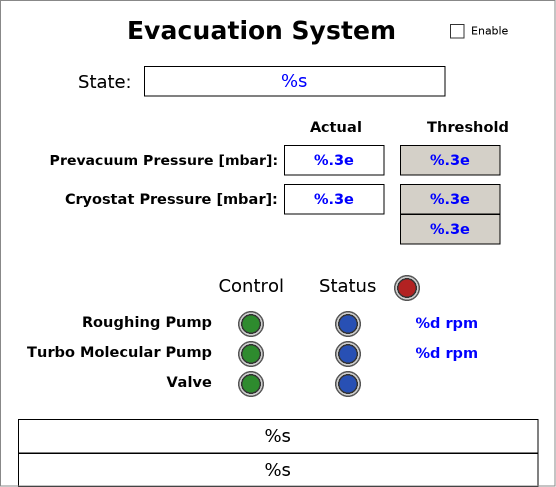
VISUALIZATION GUI_TEMPLATE_CRYO_EVAC_BASE  // 556x487
VAR_IN_OUT
	m_Instance:	FB_CRYO_EVAC_BASE;
	m_bEnable:	BOOL;
END_VAR
    Rectangle (144,66 301x30), "%s", text variable: m_Instance.stat.sState
    Lamp1 (236,309 30x30), variable: m_Instance.ctrl.bEnable_RP, style: Lamp-Lamp1-Green
    Rectangle (15,307 200x30), "Roughing Pump"
    Lamp1 (236,339 30x30), variable: m_Instance.ctrl.bEnable_TP, style: Lamp-Lamp1-Green
    Rectangle (15,337 200x30), "Turbo Molecular Pump"
    Lamp1 (236,369 30x30), variable: m_Instance.ctrl.bEnable_Valve, style: Lamp-Lamp1-Green
    Rectangle (15,367 200x30), "Valve"
    Rectangle (18,419 520x34), "%s", tooltip "Error description", text variable: m_Instance.stat.sErrorText
    Checkbox (448,16 108x30), "Enable", variable: m_bEnable
    Rectangle (56,67 84x30), "State:"
    Rectangle (299,271 98x30), "Status"
    Rectangle (284,145 100x30), "%.3e", tooltip "Prevacuum pressure [mbar]", text variable: m_Instance.prevac.stat.lrPressure
    Rectangle (400,145 100x30), "%.3e", tooltip "Prevacuum pressure threshold [mbar]", text variable: m_Instance.cfg.lrThld_Prevac
    Rectangle (284,184 100x30), "%.3e", tooltip "Cryo pressure [mbar]", text variable: m_Instance.in_lrCryoPressure
    Rectangle (400,184 100x30), "%.3e", tooltip "Pressure threshold for safe start of Turbo Pump [mbar]", text variable: m_Instance.cfg.lrThld_TP_SafeStartPressure
    Rectangle (400,214 100x30), "%.3e", tooltip "Pressure threshold for safe opening of the pre-vacuum valve [mbar]", text variable: m_Instance.cfg.lrThld_Valve_SafeOpenPressure
    Rectangle (51,145 230x30), "Prevacuum Pressure [mbar]:"
    Rectangle (51,184 230x30), "Cryostat Pressure [mbar]:"
    Rectangle (307,112 232x30), "Actual Threshold"
    Lamp1 (333,309 30x30), tooltip "If ON, Pump is Running", variable: m_Instance.stat.bRootPumpON, style: Lamp-Lamp1-Blue
    Lamp1 (333,339 30x30), tooltip "If ON, Pump is Running", variable: m_Instance.stat.bTurboPumpON, style: Lamp-Lamp1-Blue
    Lamp1 (333,369 30x30), tooltip "If ON, Insulation Valve is OPEN", variable: m_Instance.valve.stat.bActON, style: Lamp-Lamp1-Blue
    Rectangle (381,308 100x30), "%d rpm", tooltip "Roughing Pump Speed [rpm]", text variable: m_Instance.rpRef.statBaseRef.nPumpSpeed
    Rectangle (381,338 100x30), "%d rpm", tooltip "Turbo Pump Speed [rpm]", text variable: m_Instance.tp.stat.nPumpSpeed
    Rectangle (92,13 339x34), "Evacuation System"
    Rectangle (195,271 113x30), "Control"
    Rectangle (18,453 520x34), "%s", tooltip "Evacuation System Status", text variable: m_Instance.stat.sStatus
    Lamp1 (392,273 30x30), tooltip "If ON, there was an error", variable: m_Instance.stat.bError, style: Lamp-Lamp1-Red
END_VISUALIZATION

(* stored: Version 1.1.0.1, ProductVersion 3.1.4024.9
   Visu GUI_TEMPLATE_CRYO_EVAC_BASE: Id {3f948c0f-d395-40ab-be8c-d3f5b7399f7b} *)
